(* Empties/Clears/Deletes every item on the queue*)
METHOD Clear
IF THIS^.NullReferenceException() THEN RETURN; END_IF
THIS^.ipList.Clear();
END_METHOD

(* Gets and remove item at the front of the queue *)
METHOD Dequeue : I_Queue
VAR_INPUT
	Item : ANY; (* Variable to store returned item value *)
END_VAR
VAR_OUTPUT
	bSuccess : BOOL;
END_VAR
VAR 
	bA, bB 	 : BOOL;
END_VAR
Dequeue := THIS^;
IF THIS^.NullReferenceException() THEN RETURN; END_IF
THIS^.ipList.Get_First(Item, bSuccess => bA);
THIS^.ipList.Remove(bSuccess => bB);
bSuccess := bA AND bB;
END_METHOD

(* Removes item at the front of the queue without returning anything *)
METHOD Dequeue_Void : I_Queue
VAR_OUTPUT
	bSuccess : BOOL;
END_VAR
Dequeue_Void := THIS^;
IF THIS^.NullReferenceException() THEN RETURN; END_IF
THIS^.ipList.Remove(bSuccess => bSuccess);
THIS^.CatchError();
END_METHOD

(* Adds item at the back of the queue *)
METHOD Enqueue : I_Queue
VAR_INPUT
	Item : ANY; (* Variable containg data to store on the queue *)
END_VAR
VAR_OUTPUT
	bSuccess : BOOL;
END_VAR
Enqueue := THIS^;
IF THIS^.NullReferenceException() THEN RETURN; END_IF
THIS^.ipList.Add_Back(Item, bSuccess => bSuccess);
THIS^.CatchError();
END_METHOD

(* Adds item at the front of the queue *)
METHOD Enqueue_At_Front : I_Queue
VAR_INPUT
	Item : ANY; (* Variable containg data to store on the queue *)
END_VAR
VAR_OUTPUT
	bSuccess : BOOL;
END_VAR
Enqueue_At_Front := THIS^;
IF THIS^.NullReferenceException() THEN RETURN; END_IF
THIS^.ipList.Add_Front(Item, bSuccess => bSuccess);
THIS^.CatchError();
END_METHOD

(* Get item from the queue without removing it. *)
METHOD Peek : I_Queue
VAR_INPUT
	Item 	: ANY; (* Variable to store returned item value *)
	nIndex 	: DINT; (* Location of item*)
END_VAR
VAR_OUTPUT
	bSuccess : BOOL;
END_VAR
Peek := THIS^;
IF THIS^.NullReferenceException() THEN RETURN; END_IF
THIS^.ipList.Get(Item, nIndex, bSuccess => bSuccess);
THIS^.CatchError();
END_METHOD

METHOD Reverse : I_Queue
VAR_OUTPUT
	bSuccess : BOOL;
END_VAR
Reverse := THIS^;
IF THIS^.NullReferenceException() THEN RETURN; END_IF
THIS^.ipList.Reverse(bSuccess => bSuccess);
THIS^.CatchError();
END_METHOD

END_FUNCTION_BLOCK

// POUs/Examples/P_Example_List
PROGRAM INTERNAL P_Example_List
VAR
	eState 		: (IDLE, INSERT, REVERSE, RESIZE, GET, SET, FIND, CLEAR, ADD_FRONT, ADD_BACK, REMOVE, REMOVE_AT);
	fbList 		: FB_List;
	nFind 		: DINT;
	sData 		: WSTRING;
	sRTNData	: ARRAY[0..6] OF WSTRING;
	nCount 		: DINT;
	stError 	: ST_ERROR;
END_VAR

stError := fbList._Error_Status;
CASE eState OF
	INSERT:
		sData := "Cats";	fbList.Insert(sData, 0);
		sData := "Dogs";	fbList.Insert(sData, 1);
		sData := "Ravens";	fbList.Insert(sData, 2);
		sData := "Mollies";	fbList.Insert(sData, 3);
	REVERSE:
		fbList.Reverse();
	RESIZE:
		fbList.Resize(3);
	GET: 
		Scrub();
		fbList
			.Get(sRTNData[0], 0)
			.Get(sRTNData[1], 1)
			.Get(sRTNData[2], 2)
			.Get(sRTNData[3], 3)
			.Get(sRTNData[4], 4)
			.Get(sRTNData[5], 5)
			.Get(sRTNData[6], 6);
	SET:
		sData := "Ravens";	fbList.Set(sData, 0);
		sData := "Mollies";	fbList.Set(sData, 1);
		sData := "Dogs";	fbList.Set(sData, 2);
		sData := "Cats";	fbList.Set(sData, 3);
	FIND:
		sData := "Dogs"; fbList.Find(sData, nIndex => nFind);
	CLEAR:
		fbList.Clear();
	ADD_FRONT:
		sData := "Pythons";fbList.Add_Front(sData);
	ADD_BACK:
		sData := "Anacondas"; fbList.Add_Back(sData);
	REMOVE:
		fbList.Remove();
	REMOVE_AT:
		fbList.Remove_At(2);
END_CASE
nCount := fbList._Count;
eState := IDLE;

METHOD PRIVATE Scrub
VAR
	i 			: T_Capacity;
END_VAR
FOR i := 0 TO SIZEOF(sRTNData)/SIZEOF(sRTNData[0])-1 DO sRTNData[i] := ""; END_FOR
END_METHOD

END_PROGRAM

// POUs/Examples/P_Example_Queue
// Login into PLC and live write eState. Try nData and nRTNData once your done. eState Initialises at IDLE
PROGRAM INTERNAL P_Example_Queue
VAR
	fbList 		: FB_List;
	fbQueue 	: FB_Queue;
	sData 		: STRING;
	sRTNData	: ARRAY[0..3] OF STRING; //returned data
	nData 		: DINT;
	nRTNData 	: ARRAY[0..3] OF DINT; 
	nCount 		: DINT;
	eState 		: (IDLE, ENQUEUE_AND_PEEK, GET_ITEM_COUNT,REVERSE_AND_PEEK, DEQUEUE_AND_PEEK, CLEAR_Q);
	stError 	: ST_ERROR;
END_VAR

fbQueue(ipList := fbList);
stError := fbQueue._Error_Status;
CASE eState OF
	ENQUEUE_AND_PEEK: //
		sData := 'Cats';fbQueue.Enqueue(sData);
		sData := 'Dogs';fbQueue.Enqueue(sData);
		sData := 'Birds';fbQueue.Enqueue(sData);
		sData := 'Fish';fbQueue.Enqueue_At_Front(sData);

		fbQueue.Peek(sRTNData[0], 0)
			   .Peek(sRTNData[1], 1)
			   .Peek(sRTNData[2], 2)
			   .Peek(sRTNData[3], 3);
		eState := IDLE;
		
	GET_ITEM_COUNT: 
		nCount := fbQueue._Count;
		eState := IDLE;
		
	REVERSE_AND_PEEK:
		fbQueue.Reverse()
			   .Peek(sRTNData[0], 0)
			   .Peek(sRTNData[1], 1)
			   .Peek(sRTNData[2], 2)
			   .Peek(sRTNData[3], 3);
		eState := IDLE;
	
	DEQUEUE_AND_PEEK:
		fbQueue.Dequeue(sRTNData[0])
			   .Dequeue_Void()
			   .Peek(sRTNData[1], 1)
			   .Peek(sRTNData[2], 2)
			   .Peek(sRTNData[3], 3);
		eState := IDLE;
		
	CLEAR_Q:
		fbQueue.Clear();
		eState := IDLE;	
END_CASE

END_PROGRAM

// POUs/Examples/P_Example_Stack
// Login into PLC and live write eState. Try nData and nRTNData once your done. eState Initialises at IDLE
PROGRAM INTERNAL P_Example_Stack
VAR
	fbList 		: FB_List;
	fbStack 	: FB_Stack;
	sData 		: STRING;
	sRTNData	: ARRAY[0..3] OF STRING; //returned data
	nData 		: DINT;
	nRTNData 	: ARRAY[0..3] OF DINT; 
	nCount 		: DINT;
	eState 		: (IDLE, PUSH_AND_PEEK, GET_ITEM_COUNT,REVERSE_AND_PEEK, POP, CLEAR_STACK);
	stError 	: ST_ERROR;
END_VAR

fbStack(ipList := fbList);
stError := fbStack._Error_Status;
CASE eState OF
	PUSH_AND_PEEK:
		sData := 'Cats';fbStack.Push(sData);
		sData := 'Dogs';fbStack.Push(sData);
		sData := 'Birds';fbStack.Push(sData);
		sData := 'Fish';fbStack.Push(sData);

		fbStack.Peek(sRTNData[0], 0)
			   .Peek(sRTNData[1], 1)
			   .Peek(sRTNData[2], 2)
			   .Peek(sRTNData[3], 3);
		eState := IDLE;
		
	GET_ITEM_COUNT: 
		nCount := fbStack._Count;
		eState := IDLE;
		
	REVERSE_AND_PEEK:
		fbStack.Reverse()
			   .Peek(sRTNData[0], 0)
			   .Peek(sRTNData[1], 1)
			   .Peek(sRTNData[2], 2)
			   .Peek(sRTNData[3], 3);
		eState := IDLE;
	
	POP:
		fbStack.Pop(sRTNData[0])
			   .Pop(sRTNData[1])
			   .Pop(sRTNData[2]);
		eState := IDLE;
		
	CLEAR_STACK:
		fbStack.Clear();
		eState := IDLE;	
END_CASE

END_PROGRAM

// POUs/Examples/P_Example_Tree_Map
PROGRAM INTERNAL P_Example_Tree_Map
VAR
	sz 			: UDINT;
	eState 		: (IDLE, TRAVERSE, INSERT, GET, UPDATE, REMOVE, CLEAR, BALANCE);
	eTrav 		: T_BST_Traversal;
	fbTree_Map	: FB_Tree_Map;
	arUpdate 	: ARRAY[0..1] OF WSTRING := ["Python", ""];
	arKeys		: ARRAY[0..6] OF WSTRING := ["qwerty","play","thomas","jerry",   "perry",    "sarah"];
	arValues	: ARRAY[0..6] OF WSTRING := ["Cats",  "Dogs","Ravens","Mollies", "Anaconda", "cow"];
	arRTNData	: ARRAY[0..6] OF WSTRING;
	arTravData 	: ARRAY[0..1] OF ARRAY[0..9] OF STRING;
	rmvdVal,
	Key, 
	Value		: WSTRING;
	nCount,i 	: DINT;
	stError 	: ST_ERROR;
END_VAR

stError := fbTree_Map._Error_Status;
sz := SIZEOF(fbTree_Map);
nCount := fbTree_Map._Count;
CASE eState OF
	INSERT:
		fbTree_Map
			.Insert(arKeys[0], arValues[0])
			.Insert(arKeys[1], arValues[1])
			.Insert(arKeys[2], arValues[2])
			.Insert(arKeys[3], arValues[3])
			.Insert(arKeys[4], arValues[4])
			.Insert(arKeys[5], arValues[5]);
	GET:
		Scrub();
		fbTree_Map
			.Get(arKeys[0], arRTNData[0])
			.Get(arKeys[1], arRTNData[1])
			.Get(arKeys[2], arRTNData[2])
			.Get(arKeys[3], arRTNData[3])
			.Get(arKeys[4], arRTNData[4])
			.Get(arKeys[5], arRTNData[5]);
			
	TRAVERSE:
		fbTree_Map._Traversal := eTrav;
		FOR i := 0 TO fbTree_Map._Keys._Count-1 DO 
			arTravData[0][i] := ''; // Key
			arTravData[1][i] := ''; // Value
			fbTree_Map._Keys.Get_Value_As_String(i, sItem => arTravData[0][i]);
			fbTree_Map._Values.Get_Value_As_String(i, sItem => arTravData[1][i]); 
			END_FOR
			
	UPDATE:
		fbTree_Map.Update(arKeys[1], arUpdate[0]);
		
	REMOVE:
		fbTree_Map.Get(arKeys[3],rmvdVal).Remove(arKeys[3]);
 
	CLEAR:
		fbTree_Map.Clear();
		
	BALANCE:
		fbTree_Map.Balance();
END_CASE
eState := IDLE;

METHOD PRIVATE Scrub
VAR
	i 			: T_Capacity;
END_VAR
FOR i := 0 TO SIZEOF(arRTNData)/SIZEOF(arRTNData[0])-1 DO arRTNData[i] := ""; END_FOR
END_METHOD

END_PROGRAM

// POUs/Function Blocks/FB_Tree_Map
// Binary search tree based map
{attribute 'enable_dynamic_creation'}
FUNCTION_BLOCK FB_Tree_Map EXTENDS FB_Collection IMPLEMENTS I_Tree_Map
VAR
	pRoot 			 		: POINTER TO ST_TREE_MAP_ENTRY_NODE;
	eTraversal 		 		: T_BST_Traversal;
	pKey_List,
	pValue_List 	 		: POINTER TO FB_List;
	pRead_Only_Key_List,
	pRead_Only_Value_List 	: POINTER TO FB_Read_Only_List;
END_VAR

// Checks if bst is ready to be balanced
METHOD PROTECTED Balance_Ready : BOOL
VAR
	nMod 		: T_Capacity;
END_VAR
VAR CONSTANT
	nMod_Const 	: T_Capacity := 4; 
END_VAR
nMod := THIS^._Count MOD nMod_Const;
Balance_Ready := nMod = 0;
END_METHOD

// Compare A to B -> A<B = -1, A=B = 0, A>B = 1
METHOD PROTECTED Compare : DINT
VAR_INPUT
	A, B 	: T_Generic;
END_VAR
VAR
	nSizeA, 
	nSizeB 	: UDINT;
	n 		: DINT; 
END_VAR
CASE A.TypeClass OF
	T_Type.TYPE_STRING:
		nSizeA := LEN2(A.pValue);

	T_Type.TYPE_WSTRING:
		nSizeA := WLEN2(A.pValue);
ELSE
	nSizeA := TO_UDINT(A.diSize);
END_CASE

CASE B.TypeClass OF
	T_Type.TYPE_STRING:
		nSizeB := LEN2(B.pValue);

	T_Type.TYPE_WSTRING:
		nSizeB := WLEN2(B.pValue);
ELSE
	nSizeB := TO_UDINT(B.diSize);
END_CASE

Compare := MEMCMP(A.pValue, B.pValue, MIN(nSizeA, nSizeB));
END_METHOD

// Copies A to B
METHOD PROTECTED Copy_Value : BOOL
VAR_INPUT
END_VAR
END_METHOD

METHOD PROTECTED Internal_Get
VAR_INPUT
	Key, 
	Return_Value 		: T_Generic; // Data to insert
END_VAR
VAR_OUTPUT
	bSuccess 			: BOOL; // Indicates whether operation was successful. Success = TRUE, Failure = FALSE
END_VAR
VAR
	nState 				: DINT;
	pNew_Node,
	pCurrent			: POINTER TO ST_TREE_MAP_ENTRY_NODE;
	nReturn_Value_Size,
	nValue_Size 		: UDINT;
END_VAR
IF THIS^.pRoot = 0 THEN RETURN; END_IF

pCurrent := THIS^.pRoot;
WHILE pCurrent <> 0 DO
	nState := THIS^.Compare(Key, pCurrent^.Key);
	CASE nState OF
	-1: // Less than
		pCurrent := pCurrent^.pLeft;
	 1: // Greater than
		pCurrent := pCurrent^.pRight;
	 0: // Equal
	 	IF Return_Value.TypeClass <> pCurrent^.Value.TypeClass THEN RETURN; END_IF
		CASE Return_Value.TypeClass OF
			T_Type.TYPE_STRING: 
				nReturn_Value_Size 	:= LEN2(Return_Value.pValue)+1;
				nValue_Size 		:= LEN2(pCurrent^.Value.pValue)+1;
			T_Type.TYPE_WSTRING:
				nReturn_Value_Size 	:= (WLEN2(Return_Value.pValue)*SIZEOF(WORD))+SIZEOF(WORD);
				nValue_Size 		:= (WLEN2(pCurrent^.Value.pValue)*SIZEOF(WORD))+SIZEOF(WORD);
		ELSE
			IF Return_Value.diSize <> pCurrent^.Value.diSize THEN RETURN; END_IF
			nReturn_Value_Size 		:= TO_UDINT(Return_Value.diSize);
			nValue_Size 			:= TO_UDINT(pCurrent^.Value.diSize);
		END_CASE
		MEMMOVE(Return_Value.pValue, pCurrent^.Value.pValue, nValue_Size);
		bSuccess := TRUE;
	 	EXIT; 
	ELSE
		EXIT;
	END_CASE
	END_WHILE
END_METHOD

METHOD PROTECTED Internal_Insert
VAR_INPUT
	Key, Value 		: T_Generic; // Data to insert
END_VAR
VAR_OUTPUT
	bSuccess 	: BOOL; // Indicates whether operation was successful. Success = TRUE, Failure = FALSE
END_VAR
VAR
	nState 		: DINT;
	pNew_Node,
	pCurrent	: POINTER TO ST_TREE_MAP_ENTRY_NODE;
END_VAR
pNew_Node := THIS^.Malloc_Node(Key, Value);

IF THIS^.pRoot = 0 THEN THIS^.pRoot := pNew_Node; bSuccess := TRUE; THIS^.IncrementCount(); RETURN; END_IF

pCurrent := THIS^.pRoot;
WHILE pCurrent <> 0 DO
	nState := THIS^.Compare(Key, pCurrent^.Key);
	CASE nState OF
	-1: // Less than
		IF pCurrent^.pLeft = 0 THEN pCurrent^.pLeft  := pNew_Node; bSuccess := TRUE; THIS^.IncrementCount(); RETURN; END_IF
		pCurrent  := pCurrent^.pLeft;
	 1: // Greater than
		IF pCurrent^.pRight = 0 THEN pCurrent^.pRight := pNew_Node; bSuccess := TRUE; THIS^.IncrementCount(); RETURN; END_IF
		pCurrent := pCurrent^.pRight;
	ELSE
		__DELETE(pNew_Node^.Key.pValue);
		__DELETE(pNew_Node^.Value.pValue);
		__DELETE(pNew_Node);
		EXIT;
	END_CASE
	END_WHILE
END_METHOD

METHOD PROTECTED Internal_Remove : POINTER TO T_BST_Node
VAR_INPUT
	Key				: T_Generic; 	// Data to remove
END_VAR
VAR_OUTPUT
	bSuccess 		: BOOL; 		// Indicates whether operation was successful. Success = TRUE, Failure = FALSE
END_VAR
VAR
	nState, nFirst 	: DINT;
	pCurrent, 
	pParent,
	pChild,
	pMin			: POINTER TO ST_TREE_MAP_ENTRY_NODE;
	bInit 			: BOOL := TRUE;
END_VAR
pCurrent := THIS^.pRoot;
WHILE pCurrent <> 0 DO
	nState := THIS^.Compare(Key, pCurrent^.Key);
	IF bInit THEN nFirst := nState; bInit := FALSE; END_IF
	CASE nState OF
	 0: // Equal
	 	EXIT;
	-1: // Less than
		pParent := pCurrent; pCurrent := pCurrent^.pLeft;
	 1: // Greater than   
	 	pParent := pCurrent; pCurrent := pCurrent^.pRight;
	END_CASE
	END_WHILE

IF pCurrent = 0 THEN RETURN; END_IF // Return if node not found

bSuccess := TRUE;
THIS^.DecrementCount();
 
IF (pCurrent^.pLeft = 0) OR (pCurrent^.pRight = 0) THEN
	
	pChild := SEL(pCurrent^.pLeft = 0, pCurrent^.pLeft, pCurrent^.pRight);
	
	IF pParent = 0 THEN 
		THIS^.pRoot := pChild;
	ELSE 
		IF pCurrent = pParent^.pLeft THEN pParent^.pLeft := pChild; ELSE pParent^.pRight := pChild; END_IF
		END_IF
		
	__DELETE(pCurrent^.Key.pValue);
	__DELETE(pCurrent^.Value.pValue);
 	__DELETE(pCurrent);
	RETURN;
	END_IF
	
pParent := pCurrent;
pMin 	:= pCurrent^.pRight;
WHILE (pMin^.pLeft <> 0) DO
	pParent := pMin;
	pMin 	:= pMin^.pLeft;
	END_WHILE

pCurrent^.Key := pMin^.Key;
pCurrent^.Value := pMin^.Value;
IF pMin = pParent^.pLeft THEN pParent^.pLeft := pMin^.pRight; ELSE pParent^.pRight := pMin^.pRight; END_IF

__DELETE(pMin^.Key.pValue);
__DELETE(pMin^.Value.pValue);
__DELETE(pMin);
END_METHOD

(* Traveses the binary search tree and appends into a collection *)
METHOD PROTECTED Internal_Traversal
VAR_INPUT
	bValue 			: BOOL;				 // By if TRUE ipGeneric_List if populated with values else it's populated with keys 
	ipGeneric_List 	: I_Generic_List; // Collection to append data to.
END_VAR
VAR
	pList 		: POINTER TO FB_List;
	pQueue 		: POINTER TO FB_Queue;
	pStack 		: POINTER TO FB_Stack;
	pCurrent,
	pPrevious 	: POINTER TO ST_TREE_MAP_ENTRY_NODE;
END_VAR
IF THIS^.pRoot = 0 THEN RETURN; END_IF
IF ipGeneric_List = 0 THEN RETURN; END_IF

pList := __NEW(FB_List);

CASE THIS^._Traversal OF
	T_BST_Traversal.Inorder:
		// In Order Traversal
		pStack := __NEW(FB_Stack);
		pStack^(ipList := pList^);
		pCurrent := THIS^.pRoot;
		WHILE (pCurrent <> 0) OR (NOT pStack^._Is_Empty) DO
			IF pCurrent <> 0 THEN pStack^.Push(pCurrent); pCurrent := pCurrent^.pLeft; CONTINUE; END_IF
			pStack^.Pop(pCurrent); 
			
			IF bValue THEN
				ipGeneric_List.Insert_Generic(pCurrent^.Value, ipGeneric_List._Count);
			ELSE
				ipGeneric_List.Insert_Generic(pCurrent^.Key, ipGeneric_List._Count);
				END_IF
			
			pCurrent := pCurrent^.pRight;
			END_WHILE
		__DELETE(pStack);
		
	T_BST_Traversal.Postorder:
		// Post Order
		pStack := __NEW(FB_Stack);
		pStack^(ipList := pList^);
		pCurrent := THIS^.pRoot;
		
		WHILE (pCurrent <> 0) OR (NOT pStack^._Is_Empty) DO
			IF pCurrent <> 0 THEN pStack ^.Push(pCurrent); pCurrent := pCurrent^.pLeft; CONTINUE; END_IF
			pStack^.Top(pCurrent);
			IF (pCurrent^.pRight = 0) OR (pCurrent^.pRight = pPrevious) THEN
				
				IF bValue THEN
					ipGeneric_List.Insert_Generic(pCurrent^.Value, ipGeneric_List._Count);
				ELSE
					ipGeneric_List.Insert_Generic(pCurrent^.Key, ipGeneric_List._Count);
					END_IF
				
				pStack^.Pop_Void();
				pPrevious := pCurrent;
				pCurrent := 0;
				CONTINUE;
				END_IF
			pCurrent := pCurrent^.pRight;
			END_WHILE
		__DELETE(pStack);
		
	T_BST_Traversal.Preorder:
		// Preoder Traversal
		pStack := __NEW(FB_Stack);
		pStack^(ipList := pList^);
		pCurrent := THIS^.pRoot;
		pStack^.Push(pCurrent);
		WHILE NOT pStack^._Is_Empty DO
			pStack^.Pop(pCurrent);
			
			IF bValue THEN
				ipGeneric_List.Insert_Generic(pCurrent^.Value, ipGeneric_List._Count);
			ELSE
				ipGeneric_List.Insert_Generic(pCurrent^.Key, ipGeneric_List._Count);
				END_IF
			
			IF pCurrent^.pRight <> 0 THEN pStack^.Push(pCurrent^.pRight); END_IF
			IF pCurrent^.pLeft  <> 0 THEN pStack^.Push(pCurrent^.pLeft); END_IF
			END_WHILE
		__DELETE(pStack);
		
	T_BST_Traversal.Level_Order:
		// Level Traversal
		pQueue 	:= __NEW(FB_Queue);
		pQueue^(ipList := pList^);
		pQueue^.Enqueue(THIS^.pRoot);
		WHILE NOT pQueue^._Is_Empty DO
			pQueue^.Dequeue(pCurrent);
			IF pCurrent^.pLeft <> 0 THEN pQueue^.Enqueue(pCurrent^.pLeft);END_IF
			IF pCurrent^.pRight <> 0 THEN pQueue^.Enqueue(pCurrent^.pRight);END_IF
			
			IF bValue THEN
				ipGeneric_List.Insert_Generic(pCurrent^.Value, ipGeneric_List._Count);
			ELSE
				ipGeneric_List.Insert_Generic(pCurrent^.Key, ipGeneric_List._Count);
				END_IF
				
			END_WHILE
		__DELETE(pQueue);
END_CASE
__DELETE(pList);
END_METHOD

METHOD PROTECTED Internal_Update
VAR_INPUT
	Key, Value 		: T_Generic; // Data to insert
END_VAR
VAR_OUTPUT
	bSuccess 	: BOOL; // Indicates whether operation was successful. Success = TRUE, Failure = FALSE
END_VAR
VAR
	nState 		: DINT;
	pNew_Node,
	pCurrent	: POINTER TO ST_TREE_MAP_ENTRY_NODE;
END_VAR
pNew_Node := THIS^.Malloc_Node(Key, Value);
IF THIS^.pRoot = 0 THEN RETURN; END_IF

pCurrent := THIS^.pRoot;
WHILE pCurrent <> 0 DO
	nState := THIS^.Compare(Key, pCurrent^.Key);
	CASE nState OF
	-1: // Less than
		pCurrent := pCurrent^.pLeft;
	 1: // Greater than
		pCurrent := pCurrent^.pRight;
	 0: // Equal
	 	__DELETE(pCurrent^.Value.pValue);
		pCurrent^.Value := THIS^.Malloc_Value(Value);
		bSuccess := TRUE;
	 	EXIT; 
	ELSE
		EXIT;
	END_CASE
	END_WHILE
END_METHOD

METHOD PROTECTED Malloc_Node : POINTER TO ST_TREE_MAP_ENTRY_NODE
VAR_INPUT
	Key, Value : T_Generic;
END_VAR
Malloc_Node 		:= __NEW(ST_TREE_MAP_ENTRY_NODE);
Malloc_Node^.Key 	:= THIS^.Malloc_Value(Key);
Malloc_Node^.Value 	:= THIS^.Malloc_Value(Value);
END_METHOD

METHOD PROTECTED Malloc_Value : T_Generic
VAR_INPUT
	Data : T_Generic;
END_VAR
// Malloc Value
Malloc_Value.TypeClass 	:= Data.TypeClass;
Malloc_Value.diSize 	:= Data.diSize;
Malloc_Value.pValue 	:= __NEW(BYTE, TO_UDINT(Data.diSize));
MEMMOVE(Malloc_Value.pValue, Data.pValue, TO_UDINT(Data.diSize));
END_METHOD

// Gets a read-only list of the keys
PROPERTY _Keys : I_Read_Only_List
GET
IF THIS^.pKey_List = 0 THEN THIS^.pKey_List := __NEW(FB_List); END_IF
IF THIS^.pRead_Only_Key_List = 0 THEN THIS^.pRead_Only_Key_List := __NEW(FB_Read_Only_List); END_IF

THIS^.pKey_List^.Clear();
THIS^.Internal_Traversal(FALSE,THIS^.pKey_List^);

THIS^.pRead_Only_Key_List^(ipList := THIS^.pKey_List^);
_Keys := THIS^.pRead_Only_Key_List^;
END_GET
END_PROPERTY

// Get and set the order in which the property _Keys/Value should return values
PROPERTY _Traversal : T_BST_Traversal
GET
_Traversal := THIS^.eTraversal;
END_GET
SET
THIS^.eTraversal := _Traversal;
END_SET
END_PROPERTY

// Gets a read-only list of the values
PROPERTY _Values : I_Read_Only_List
GET
IF THIS^.pValue_List = 0 THEN THIS^.pValue_List := __NEW(FB_List); END_IF
IF THIS^.pRead_Only_Value_List = 0 THEN THIS^.pRead_Only_Value_List := __NEW(FB_Read_Only_List); END_IF

THIS^.pValue_List^.Clear();
THIS^.Internal_Traversal(TRUE,THIS^.pValue_List^);

THIS^.pRead_Only_Value_List^(ipList := THIS^.pValue_List^);
_Values := THIS^.pRead_Only_Value_List^;
END_GET
END_PROPERTY

// Balances Tree Map. Tree will normal auto balance every time its count is a multiple of 4
METHOD Balance
VAR
	pTemp 			 	 : POINTER TO ST_TREE_MAP_ENTRY_NODE;
	pStack 				 : POINTER TO FB_Stack;
	pStack_List,
	pOrdered_List 		 : POINTER TO FB_List;
	pHelper_BST_Balancer : POINTER TO FB_Helper_Tree_Map_Balancer;
END_VAR
IF THIS^.pRoot = 0 THEN RETURN; END_IF

// Create helpers
pHelper_BST_Balancer := __NEW(FB_Helper_Tree_Map_Balancer);
pStack_List 		 := __NEW(FB_List);
pOrdered_List 		 := __NEW(FB_List);
pStack 				 := __NEW(FB_Stack);
pStack^(ipList := pStack_List^);

// Inorder traversal
pTemp := THIS^.pRoot;
WHILE (pTemp <> 0) OR (NOT pStack^._Is_Empty) DO
	IF pTemp <> 0 THEN pStack^.Push(pTemp); pTemp := pTemp^.pLeft; CONTINUE; END_IF
	pStack^.Pop(pTemp); 
	pOrdered_List^.Add_Back(pTemp);
	pTemp := pTemp^.pRight;
	END_WHILE

// Balance BST
pTemp := 0;
pHelper_BST_Balancer^(ipList := pOrdered_List^, nStart := 0, nEnd := pOrdered_List^._Count -1 , pNode => pTemp);
IF pTemp <> 0 THEN THIS^.pRoot := pTemp; END_IF

pStack_List^.Clear();

// Delete helpers
__DELETE(pHelper_BST_Balancer);
__DELETE(pStack_List);
__DELETE(pStack);
__DELETE(pOrdered_List);











(*
pCurrent := THIS^.pRoot;
WHILE pCurrent <> 0 DO 
	IF pCurrent^.pLeft = 0 THEN pCurrent := pCurrent^.pRight;  CONTINUE; END_IF
	
	pPrevious := pCurrent^.pLeft;
	WHILE (pPrevious^.pRight <> 0 ) AND (pPrevious^.pRight <> pCurrent) DO
		pPrevious := pPrevious^.pRight;
		IF pPrevious^.pRight = 0 THEN pPrevious^.pRight := pCurrent; pCurrent := pCurrent^.pLeft; CONTINUE; END_IF
		pPrevious^.pRight := 0;
		pCurrent := pCurrent^.pRight;
		END_WHILE
	
	END_WHILE
*)
END_METHOD

(* Empties/Clears/Deletes every item in the collection*)
METHOD Clear
VAR
	pList 	: POINTER TO FB_List;
	pQueue 	: POINTER TO FB_Queue;
	pTemp 	: POINTER TO ST_TREE_MAP_ENTRY_NODE;
END_VAR
IF THIS^.pRoot = 0 THEN RETURN; END_IF
pList 	:= __NEW(FB_List);
pQueue 	:= __NEW(FB_Queue);
pQueue^(ipList := pList^);

pQueue^.Enqueue(THIS^.pRoot);
WHILE NOT pQueue^._Is_Empty DO
	pQueue^.Dequeue(pTemp);
	IF pTemp^.pLeft <> 0 THEN pQueue^.Enqueue(pTemp^.pLeft);END_IF
	IF pTemp^.pRight <> 0 THEN pQueue^.Enqueue(pTemp^.pRight);END_IF
	
	__DELETE(pTemp^.Key.pValue);
	__DELETE(pTemp^.Value.pValue);
	__DELETE(pTemp);
	THIS^.DecrementCount();
	END_WHILE

THIS^.pRoot := 0;
__DELETE(pQueue);
__DELETE(pList);

IF THIS^.pKey_List <> 0 THEN THIS^.pKey_List^.Clear(); END_IF
IF THIS^.pValue_List <> 0 THEN THIS^.pValue_List^.Clear(); END_IF

IF THIS^.pRead_Only_Key_List <> 0 THEN THIS^.pRead_Only_Key_List^.Clear(); END_IF
IF THIS^.pRead_Only_Value_List <> 0 THEN THIS^.pRead_Only_Value_List^.Clear(); END_IF
END_METHOD

METHOD FB_exit : BOOL
VAR_INPUT
	bInCopyCode : BOOL; // if TRUE, the exit method is called for exiting an instance that is copied afterwards (online change).
END_VAR
THIS^.Clear();
IF THIS^.pKey_List 	 <> 0 	THEN __DELETE(THIS^.pKey_List); END_IF
IF THIS^.pValue_List <> 0 	THEN  __DELETE(THIS^.pValue_List); END_IF

IF THIS^.pRead_Only_Key_List   <> 0 THEN  __DELETE(THIS^.pRead_Only_Key_List); END_IF
IF THIS^.pRead_Only_Value_List <> 0 THEN  __DELETE(THIS^.pRead_Only_Value_List); END_IF
END_METHOD

// Gets the value associated with the specified key without removing the entry from the map
METHOD Get : I_Map
VAR_INPUT
	Key 			: ANY; // Key used to identify stored value
	Return_Value 	: ANY; // Variable to store requested value 
END_VAR
VAR_OUTPUT
	bSuccess : BOOL;
END_VAR
Get := THIS^;
THIS^.Internal_Get(Key, Return_Value, bSuccess => bSuccess);
END_METHOD

// Insert an element with the provided key and value to the map
METHOD Insert : I_Map
VAR_INPUT
	Key 		: ANY; // Key used to identify stored value
	Value 		: ANY; // Value to store in map with key
END_VAR
VAR_OUTPUT
	bSuccess : BOOL;
END_VAR
Insert := THIS^;
THIS^.Internal_Insert(Key, Value, bSuccess => bSuccess);
IF NOT THIS^.Balance_Ready() THEN RETURN; END_IF
THIS^.Balance();
END_METHOD

// Removes value with the specified key from the map
METHOD Remove : I_Map
VAR_INPUT
	Key : ANY; // Key used to identify stored value
END_VAR
VAR_OUTPUT
	bSuccess : BOOL;
END_VAR
Remove := THIS^;
THIS^.Internal_Remove(Key, bSuccess => bSuccess);
IF NOT THIS^.Balance_Ready() THEN RETURN; END_IF
THIS^.Balance();
END_METHOD

// Updates the value an element with the provided key and value in the map
METHOD Update : I_Map
VAR_INPUT
	Key 	: ANY; // Key used to identify stored value
	Value 	: ANY; // Value to store in map with key
END_VAR
VAR_OUTPUT
	bSuccess : BOOL;
END_VAR
Update := THIS^;
THIS^.Internal_Update(Key, Value, bSuccess => bSuccess);
END_METHOD

END_FUNCTION_BLOCK

// POUs/Function Blocks/FB_Read_Only_List
// Read Only Decorator for function blocks that impliment I_List interface
{attribute 'enable_dynamic_creation'}
FUNCTION_BLOCK FB_Read_Only_List EXTENDS FB_Collection IMPLEMENTS I_Read_Only_List
VAR_INPUT
	ipList : I_List;
END_VAR

METHOD PROTECTED NullReferenceException : BOOL
NullReferenceException := THIS^.ipList = 0;
IF NOT NullReferenceException THEN RETURN; END_IF
THIS^.RaiseException(2000+GVL_CmpErrors.ERR_INVALID_REFERENCE, 'Null or Invalid Reference');
END_METHOD

(* Number of items in the collection*)
PROPERTY _Count : T_Capacity
GET
IF THIS^.NullReferenceException() THEN _Count := -1; RETURN; END_IF
_Count := THIS^.ipList._Count;
END_GET
END_PROPERTY

PROPERTY _Error_Status : ST_ERROR
GET
IF THIS^.NullReferenceException() THEN _Error_Status := THIS^.stError; RETURN; END_IF
THIS^.stError := THIS^.ipList._Error_Status;
_Error_Status := F_Error(THIS^.stError.bSTATUS, THIS^.stError.nCODE, THIS^.stError.sSOURCE);
END_GET
END_PROPERTY

(* Checks if collection is empty*)
PROPERTY _Is_Empty : BOOL
GET
IF THIS^.NullReferenceException() THEN _Is_Empty := TRUE; RETURN; END_IF
_Is_Empty := THIS^.ipList._Is_Empty;
END_GET
END_PROPERTY

(* DOES NOTHING - This is a read-only list *)
METHOD FINAL Clear
END_METHOD

(* Checks if item is contained in list *)
METHOD Contains : BOOL
VAR_INPUT
	Item : ANY; // Item to find in list
END_VAR
IF THIS^.NullReferenceException() THEN RETURN; END_IF
Contains := THIS^.ipList.Contains(Item);
END_METHOD

// Find the location of an item in list.
METHOD Find : I_Read_Only_List
VAR_INPUT
	Item 	: ANY; // Item to find in list
END_VAR
VAR_OUTPUT
	nIndex	: DINT; //Location of item in list 
	bSuccess : BOOL;
END_VAR
Find := THIS^;
IF THIS^.NullReferenceException() THEN nIndex := -1; RETURN; END_IF
THIS^.ipList.Find(Item, nIndex => nIndex, bSuccess => bSuccess);
END_METHOD

// Gets item from list at specified location without removing it
METHOD Get : I_Read_Only_List
VAR_INPUT
	Return_Item 	: ANY;  // Variable to store returned item
	nIndex 			: DINT; // Location of item
END_VAR
VAR_OUTPUT
	bSuccess : BOOL;
END_VAR
Get := THIS^;
IF THIS^.NullReferenceException() THEN RETURN; END_IF
THIS^.ipList.Get(Return_Item, nIndex, bSuccess => bSuccess);
END_METHOD

// Gets item at the front of the list 
METHOD Get_First : I_Read_Only_List
VAR_INPUT
	Return_Item 	: ANY; // Variable to store returned item
END_VAR
VAR_OUTPUT
	bSuccess : BOOL;
END_VAR
Get_First := THIS^;
IF THIS^.NullReferenceException() THEN RETURN; END_IF
THIS^.ipList.Get_First(Return_Item, bSuccess => bSuccess);
END_METHOD

// Gets item at the back of the list 
METHOD Get_Last : I_Read_Only_List
VAR_INPUT
	Return_Item 	: ANY; // Variable to store returned item
END_VAR
VAR_OUTPUT
	bSuccess : BOOL;
END_VAR
Get_Last := THIS^;
IF THIS^.NullReferenceException() THEN RETURN; END_IF
THIS^.ipList.Get_Last(Return_Item, bSuccess => bSuccess);
END_METHOD

// Returns item as a string, if type to string conversion is supported
METHOD Get_Value_As_String : I_Read_Only_List
VAR_INPUT
	nIndex	: DINT; // Location of item
END_VAR
VAR_OUTPUT
	sItem 	: T_MaxString; // Variable to store returned item
END_VAR
Get_Value_As_String := THIS^;
IF THIS^.NullReferenceException() THEN RETURN; END_IF
THIS^.ipList.Get_Value_As_String(nIndex, sItem => sItem);
END_METHOD

END_FUNCTION_BLOCK

// POUs/Function Blocks/Helpers/FB_Helper_Tree_Map_Balancer
// Helper to balance Binary Search Tree since recurssion is not supported
{attribute 'enable_dynamic_creation'}
FUNCTION_BLOCK INTERNAL FINAL FB_Helper_Tree_Map_Balancer
VAR_INPUT
	ipList 			: I_List;
	nStart,
	nEnd 			: T_Capacity;  
END_VAR
VAR_OUTPUT
	pNode 			: POINTER TO ST_TREE_MAP_ENTRY_NODE;
END_VAR
VAR
	bSuccess		: BOOL;
	nMid 			: T_Capacity;
	pTree_Balancer 	: POINTER TO FB_Helper_Tree_Map_Balancer;
END_VAR

IF ipList = 0 THEN RETURN; END_IF
IF nStart > nEnd THEN RETURN; END_IF

nMid := (nStart+nEnd)/2;
ipList.Get(pNode, nMid, bSuccess => bSuccess);
IF (NOT bSuccess) OR pNode = 0 THEN RETURN; END_IF 

pTree_Balancer := __NEW(FB_Helper_Tree_Map_Balancer);
pTree_Balancer^(ipList := ipList, nStart := nStart, nEnd := nMid-1, pNode => pNode^.pLeft);
pTree_Balancer^(ipList := ipList, nStart := nMid+1, nEnd := nEnd, 	pNode => pNode^.pRight);
__DELETE(pTree_Balancer);

END_FUNCTION_BLOCK

// POUs/Function Blocks/FB_Hash_Map
(*WARNING WORK-IN-PROGRESS*)
{warning 'DO NOT USE!'}
FUNCTION_BLOCK INTERNAL FB_Hash_Map EXTENDS FB_Collection IMPLEMENTS I_Map
VAR
END_VAR
VAR CONSTANT
	fbBucket_List : FB_Array_List(16) := ();
END_VAR

METHOD PROTECTED Populate_Bucket_List : BOOL
VAR_INPUT
	ipList : I_List;
	nCount : T_Capacity;
END_VAR
VAR
	
END_VAR
END_METHOD

METHOD FB_init : BOOL
VAR_INPUT
	bInitRetains 	: BOOL; // if TRUE, the retain variables are initialized (warm start / cold start)
	bInCopyCode 	: BOOL;  // if TRUE, the instance afterwards gets moved into the copy code (online change)
END_VAR
END_METHOD

// Gets the value associated with the specified key without remocing it from the dictionary
METHOD Get : I_Map
VAR_INPUT
	Key 			: ANY; // Key used to identify stored value
	Return_Value 	: ANY; // Variable to store requested data 
END_VAR
Get := THIS^;
END_METHOD

// Insert an element with the provided key and value to the dictionary
METHOD Insert : I_Map
VAR_INPUT
	Key 	: ANY; // Key used to identify stored value
	Value 	: ANY; // Value to store in dictionary with key
END_VAR
Insert := THIS^;
END_METHOD

// Removes value with the specified key from the dictionary and return that value
METHOD Remove : I_Map
VAR_INPUT
	Key 			: ANY; // Key used to identify stored value
	Return_Value 	: ANY; // Value to store in dictionary with key
END_VAR
Remove := THIS^;
END_METHOD

// Removes the value with the specified key from the dictionary and returns nothing
METHOD Remove_Void : I_Map
VAR_INPUT
	Key 	: ANY; // Key used to identify stored value
END_VAR
Remove_Void := THIS^;
END_METHOD

// Updates the value an element with the provided key and value in the dictionary
METHOD Update : I_Map
VAR_INPUT
	Key 	: ANY; // Key used to identify stored value
	Value 	: ANY; // Value to store in dictionary with key
END_VAR
Update := THIS^;
END_METHOD

END_FUNCTION_BLOCK

// POUs/Function Blocks/FB_Write_Only_List
// Write Only Decorator for function blocks that impliment I_List interface
{attribute 'enable_dynamic_creation'}
FUNCTION_BLOCK FB_Write_Only_List EXTENDS FB_Collection IMPLEMENTS I_Write_Only_List
VAR_INPUT
	ipList : I_List;
END_VAR

METHOD PROTECTED NullReferenceException : BOOL
NullReferenceException := THIS^.ipList = 0;
IF NOT NullReferenceException THEN RETURN; END_IF
THIS^.RaiseException(2000+GVL_CmpErrors.ERR_INVALID_REFERENCE, 'Null or Invalid Reference');
END_METHOD

(* Returns -1 as this is a write-only list *)
PROPERTY _Count : DINT
GET
_Count := -1;
END_GET
END_PROPERTY

PROPERTY _Error_Status : ST_ERROR
GET
IF THIS^.NullReferenceException() THEN _Error_Status := THIS^.stError; RETURN; END_IF
THIS^.stError := THIS^.ipList._Error_Status;
_Error_Status := F_Error(THIS^.stError.bSTATUS, THIS^.stError.nCODE, THIS^.stError.sSOURCE);
END_GET
END_PROPERTY

(* Returns FALSE as this is a write-only list *)
PROPERTY _Is_Empty : BOOL
GET
END_GET
END_PROPERTY

// Adds an item to the end of the list
METHOD Add_Back : I_Write_Only_List
VAR_INPUT
	Item 	: ANY; // Value to store in list
END_VAR
VAR_OUTPUT
	bSuccess : BOOL;
END_VAR
Add_Back := THIS^;
IF THIS^.NullReferenceException() THEN RETURN; END_IF
THIS^.ipList.Add_Back(Item, bSuccess => bSuccess);
END_METHOD

// Adds an item at the front of the list
METHOD Add_Front : I_Write_Only_List
VAR_INPUT
	Item 	: ANY; // Value to store in list
END_VAR
VAR_OUTPUT
	bSuccess : BOOL;
END_VAR
Add_Front := THIS^;
IF THIS^.NullReferenceException() THEN RETURN; END_IF
THIS^.ipList.Add_Front(Item, bSuccess => bSuccess);
END_METHOD

// Empties/Clears/Deletes every item in the collection
METHOD Clear
IF THIS^.NullReferenceException() THEN RETURN; END_IF
THIS^.ipList.Clear();
END_METHOD

// Adds new item to list at specified location, if index = 0, item will be added at the front, if index = count, item will be added at the back
METHOD Insert : I_Write_Only_List
VAR_INPUT
	Item 	: ANY;  // Item to store in list
	nIndex 	: DINT; // Location of item
END_VAR
VAR_OUTPUT
	bSuccess : BOOL;
END_VAR
Insert := THIS^;
IF THIS^.NullReferenceException() THEN RETURN; END_IF
THIS^.ipList.Insert(Item, nIndex, bSuccess => bSuccess);
END_METHOD

// Removes item at the front of the list and returns nothing
METHOD Remove : I_Write_Only_List
VAR_OUTPUT
	bSuccess : BOOL;
END_VAR
Remove := THIS^;
IF THIS^.NullReferenceException() THEN RETURN; END_IF
THIS^.ipList.Remove(bSuccess => bSuccess);
END_METHOD

// Remove item at specified location and return nothing
METHOD Remove_At : I_Write_Only_List
VAR_INPUT
	nIndex : DINT; // Location of item
END_VAR
VAR_OUTPUT
	bSuccess : BOOL;
END_VAR
Remove_At := THIS^;
IF THIS^.NullReferenceException() THEN RETURN; END_IF
THIS^.ipList.Remove_At(nIndex, bSuccess => bSuccess);
END_METHOD

// Removes item at the back of the list and returns nothing
METHOD Remove_Last : I_Write_Only_List
VAR_OUTPUT
	bSuccess : BOOL;
END_VAR
Remove_At := THIS^;
IF THIS^.NullReferenceException() THEN RETURN; END_IF
THIS^.ipList.Remove_Last(bSuccess => bSuccess);
END_METHOD

// Manually resize list. If list becomes smaller, item on higher locations will be deleted.
METHOD Resize : I_Write_Only_List
VAR_INPUT
	nSize : DINT; // New size of list.
END_VAR
VAR_OUTPUT
	bSuccess : BOOL;
END_VAR
Resize := THIS^;
IF THIS^.NullReferenceException() THEN RETURN; END_IF
THIS^.ipList.Resize(nSize, bSuccess => bSuccess);
END_METHOD

// Reverses the order of items in the list
METHOD Reverse : I_Write_Only_List
VAR_OUTPUT
	bSuccess : BOOL;
END_VAR
Reverse := THIS^;
IF THIS^.NullReferenceException() THEN RETURN; END_IF
THIS^.ipList.Reverse(bSuccess => bSuccess);
END_METHOD

// Adds new item to list in the specified location without resizing list
METHOD Set : I_Write_Only_List
VAR_INPUT
	Item 	: ANY; 	// Item to store in list
	nIndex 	: DINT; // Location of item
END_VAR
VAR_OUTPUT
	bSuccess : BOOL;
END_VAR
Set := THIS^;
IF THIS^.NullReferenceException() THEN RETURN; END_IF
THIS^.ipList.Set(Item, nIndex, bSuccess => bSuccess);
END_METHOD

END_FUNCTION_BLOCK

// POUs/MAIN
PROGRAM MAIN
VAR
END_VAR

P_Example_Array_List();
P_Example_Binary_Search_Tree();
P_Example_Tree_Map();
P_Example_List();
P_Example_Queue();
P_Example_Stack();

END_PROGRAM

// Project Information/F_GetCompany
// This function has been automatically generated from the project information.
{attribute 'signature_flag' := '1073741824'}
{attribute 'TcGenerated'}
{attribute 'no-analysis'}
FUNCTION F_GetCompany : WSTRING
VAR_INPUT
	
END_VAR

F_GetCompany := "FisoThemes";

END_FUNCTION

// Project Information/F_GetTitle
// This function has been automatically generated from the project information.
{attribute 'signature_flag' := '1073741824'}
{attribute 'TcGenerated'}
{attribute 'no-analysis'}
FUNCTION F_GetTitle : WSTRING
VAR_INPUT
	
END_VAR

F_GetTitle := "TwinCat Dynamic Collections";

END_FUNCTION

// Project Information/F_GetVersion
// This function has been automatically generated from the project information.
{attribute 'signature_flag' := '1073741824'}
{attribute 'TcGenerated'}
{attribute 'no-analysis'}
FUNCTION F_GetVersion : ST_LibVersion
VAR_INPUT
	
END_VAR

F_GetVersion.iMajor := 0;
F_GetVersion.iMinor := 3;
F_GetVersion.iBuild := 1;
F_GetVersion.iRevision := 0;

END_FUNCTION
